// TIA Portal project "ISA_P6" (V16)

(* hardware
DEVICE "SINAMICS G_1"  Sinamics.Device
   slot 0: "Accionamiento_1"  G120 CU250S-2 PN Vector  6SL3246-0BA22-1FA0  4.7.10
      slot 1: "Interfaz PROFINET"  MDD-SinamicsG120-P
   slot 0: "	_0"  Rail  SinamicsG120SVecto
   slot 3: "PM240 IP20"  PM240 IP20  6SL3224-0BE13-7UA0  -
DEVICE "S7-1200 station_1"  S7-1200 Station
   slot 0: "Rack_0"  S7-1200 Rack  Rack  V1.0
   slot 1: "PLC_1"  CPU 1215C DC/DC/DC  6ES7 215-1AG40-0XB0  V4.4
DEVICE "PC-System_1"  SIMATIC PC station
   slot 0: "Estación PC SIMATIC"  Rail  SIMATIC PC-Station  V1.0
      slot 125: "Stationmanager"  Station_Manager  V6.0.4
   slot 1: "HMI_RT_1"  WinCC RT Advanced  6AV2 104-0xxxx-xxxx  16.0.0.0
      slot 33792: "Interfaz del equipo"  Host interface
   slot 2: "IE general_1"  IE General  IE_CP  V8.2.0
*)

// ===== PLC "PLC_1"  CPU 1215C DC/DC/DC =====

VAR_GLOBAL   // PLC tag table "Tabla de variables estándar"
   "ConexiónMotor" AT %Q0.0 : Bool;
   "InversionSentido" AT %Q0.1 : Bool;
   "ConsignaVelocidad" AT %QW64 : Int;
   "ConsignaVelocidadAlcanzada" AT %I0.0 : Bool;
   "ActivarJog1" AT %Q0.2 : Bool;
   "VelocidadActual" AT %IW64 : Word;
END_VAR

DATA_BLOCK "Variables"   // DB1
{ S7_Optimized_Access := 'TRUE' }
VERSION : 0.1
   VAR
      ConexionMotorScada : Bool;
      VelocidadConsignaAlcanzadaScada : Bool;
      InversionMotorScada : Bool;
      VelocidadActualScada : Bool;
      ActivarJog1Scada : Bool;
      VelocidadMotorScada : Int;
      VelocidadNormalizada : Real;
      VelocidadEscalada : Int;
      VelocidadReal : Real;
   END_VAR
BEGIN
END_DATA_BLOCK

DATA_BLOCK "VelocidadReal"   // DB2
{ S7_Optimized_Access := 'TRUE' }
VERSION : 0.1
// stored: InstanceOfName Analog_IN
"Analog_IN"
BEGIN
END_DATA_BLOCK

DATA_BLOCK "Telerruptor_DB"   // DB3
{ S7_Optimized_Access := 'TRUE' }
VERSION : 0.1
// stored: InstanceOfName Telerruptor
"Telerruptor"
BEGIN
END_DATA_BLOCK

DATA_BLOCK "Analog_IN_1_DB"   // DB4
{ S7_Optimized_Access := 'TRUE' }
VERSION : 0.1
// stored: InstanceOfName Analog_IN_1
"Analog_IN_1"
BEGIN
END_DATA_BLOCK

DATA_BLOCK "Analog_OUT_DB"   // DB5
{ S7_Optimized_Access := 'TRUE' }
VERSION : 0.1
// stored: InstanceOfName Analog_OUT
"Analog_OUT"
BEGIN
END_DATA_BLOCK

FUNCTION_BLOCK "Telerruptor"   // FB2, LAD
{ S7_Optimized_Access := 'TRUE' }
VERSION : 0.1
   VAR_INPUT
      Pulsador : Bool;
   END_VAR
   VAR_OUTPUT
      Salida : Bool;
   END_VAR
   VAR
      Flanco : Bool;
      "on/off" : Bool;
      state : Bool;
   END_VAR
   VAR_TEMP   // added for the SCL form of the ladder/FBD networks
      _w1 : Bool;
   END_VAR
BEGIN

REGION Network 1
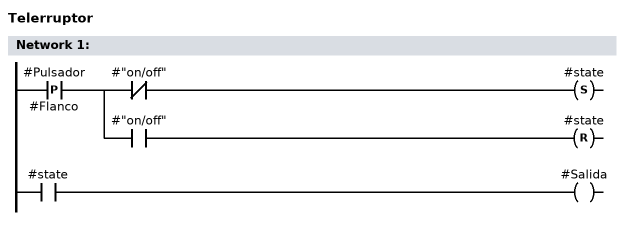
   RUNG wire#powerrail
      P_Contact(operand := #Pulsador, bit := #Flanco)
      wire#w1
      I_Contact( #"on/off" )
      S_Coil( #state )
   END_RUNG
   RUNG wire#w1
      Contact( #"on/off" )
      R_Coil( #state )
   END_RUNG
   RUNG wire#powerrail
      Contact( #state )
      Coil( #Salida )
   END_RUNG
   // the same network as SCL:
   #_w1 := #Pulsador AND NOT #Flanco;   // rising edge of #Pulsador
   #Flanco := #Pulsador;
   IF #_w1 AND NOT #"on/off" THEN #state := TRUE; END_IF;
   IF #_w1 AND #"on/off" THEN #state := FALSE; END_IF;
   #Salida := #state;
END_REGION
END_FUNCTION_BLOCK

FUNCTION_BLOCK "Analog_IN"   // FB4, LAD
{ S7_Optimized_Access := 'TRUE' }
VERSION : 0.1
   VAR_INPUT
      Input : Int;
      X_min : Real;
      X_max : Real;
      Y_min : Real;
      Y_max : Real;
      IsTension : Bool;
   END_VAR
   VAR_OUTPUT
      Output : Real;
   END_VAR
   VAR
      X_min_bits : Int;
      X_max_bits : Int;
      norm : Real;
   END_VAR
   VAR CONSTANT
      tension_pendent : Real := 2764.8;
      intensity_pendent : Real := 1382.4;
   END_VAR
BEGIN

REGION Network 1 (SCL)

   IF #IsTension THEN
       #X_min_bits := REAL_TO_INT(#X_min * #tension_pendent);
       #X_max_bits := REAL_TO_INT(#X_max * #tension_pendent);
   ELSE
       #X_min_bits := REAL_TO_INT(#X_min * #intensity_pendent);
       #X_max_bits := REAL_TO_INT(#X_max * #intensity_pendent);
   END_IF;
END_REGION

REGION Network 2
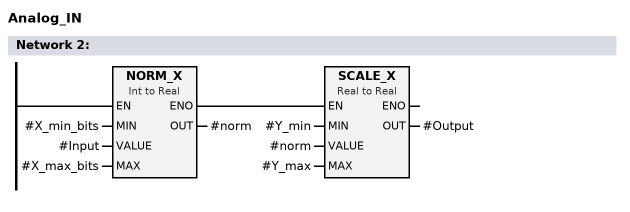
   RUNG wire#powerrail
      { S7_Templates := "[SrcType := Int, DestType := Real]" } Normalize(min := #X_min_bits, value := #Input, max := #X_max_bits, out => #norm)
      { S7_Templates := "[SrcType := Real, DestType := Real]" } Scale(min := #Y_min, value := #norm, max := #Y_max, out => #Output)
   END_RUNG
   // the same network as SCL:
   #norm := NORM_X(MIN := #X_min_bits, VALUE := #Input, MAX := #X_max_bits);
   #Output := SCALE_X(MIN := #Y_min, VALUE := #norm, MAX := #Y_max);
END_REGION
END_FUNCTION_BLOCK

FUNCTION_BLOCK "Analog_IN_1"   // FB4, LAD
{ S7_Optimized_Access := 'TRUE' }
VERSION : 0.1
   VAR_INPUT
      Input : Int;
      X_min : Real;
      X_max : Real;
      Y_min : Real;
      Y_max : Real;
      IsTension : Bool;
   END_VAR
   VAR_OUTPUT
      Output : Real;
   END_VAR
   VAR
      X_min_bits : Int;
      X_max_bits : Int;
      norm : Real;
   END_VAR
   VAR CONSTANT
      tension_pendent : Real := 2764.8;
      intensity_pendent : Real := 1382.4;
   END_VAR
BEGIN

REGION Network 1 (SCL)

   IF #IsTension THEN
       #X_min_bits := REAL_TO_INT(#X_min * #tension_pendent);
       #X_max_bits := REAL_TO_INT(#X_max * #tension_pendent);
   ELSE
       #X_min_bits := REAL_TO_INT(#X_min * #intensity_pendent);
       #X_max_bits := REAL_TO_INT(#X_max * #intensity_pendent);
   END_IF;
END_REGION

REGION Network 2
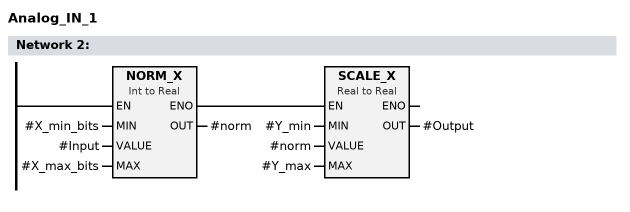
   RUNG wire#powerrail
      { S7_Templates := "[SrcType := Int, DestType := Real]" } Normalize(min := #X_min_bits, value := #Input, max := #X_max_bits, out => #norm)
      { S7_Templates := "[SrcType := Real, DestType := Real]" } Scale(min := #Y_min, value := #norm, max := #Y_max, out => #Output)
   END_RUNG
   // the same network as SCL:
   #norm := NORM_X(MIN := #X_min_bits, VALUE := #Input, MAX := #X_max_bits);
   #Output := SCALE_X(MIN := #Y_min, VALUE := #norm, MAX := #Y_max);
END_REGION
END_FUNCTION_BLOCK

FUNCTION_BLOCK "Analog_OUT"   // FB5, LAD
{ S7_Optimized_Access := 'TRUE' }
VERSION : 0.1
   VAR_INPUT
      Input : Real;
      X_min : Real;
      X_max : Real;
      Y_min : Real;
      Y_max : Real;
      IsTension : Bool;
   END_VAR
   VAR_OUTPUT
      Output : Int;
   END_VAR
   VAR
      Y_min_bits : Int;
      Y_max_bits : Int;
      norm : Real;
   END_VAR
   VAR CONSTANT
      tension_pendent : Real := 2764.8;
      intensity_pendent : Real := 1382.4;
   END_VAR
BEGIN

REGION Network 1 (SCL)

   IF #IsTension THEN
       #Y_min_bits := REAL_TO_INT(#Y_min * #tension_pendent);
       #Y_max_bits := REAL_TO_INT(#Y_max * #tension_pendent);
   ELSE
       #Y_min_bits := REAL_TO_INT(#Y_min * #intensity_pendent);
       #Y_max_bits := REAL_TO_INT(#Y_max * #intensity_pendent);
   END_IF;
END_REGION

REGION Network 2
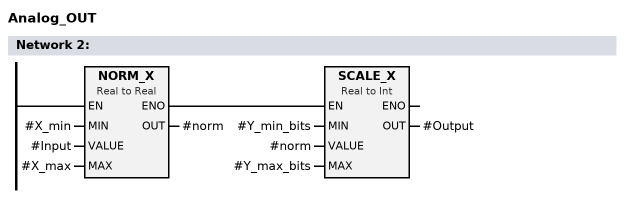
   RUNG wire#powerrail
      { S7_Templates := "[SrcType := Real, DestType := Real]" } Normalize(min := #X_min, value := #Input, max := #X_max, out => #norm)
      { S7_Templates := "[SrcType := Real, DestType := Int]" } Scale(min := #Y_min_bits, value := #norm, max := #Y_max_bits, out => #Output)
   END_RUNG
   // the same network as SCL:
   #norm := NORM_X(MIN := #X_min, VALUE := #Input, MAX := #X_max);
   #Output := SCALE_X(MIN := #Y_min_bits, VALUE := #norm, MAX := #Y_max_bits);
END_REGION
END_FUNCTION_BLOCK

ORGANIZATION_BLOCK "Variador"   // OB1, LAD, ProgramCycle
TITLE = "Main Program Sweep (Cycle)"
{ S7_Optimized_Access := 'TRUE' }
VERSION : 0.1
   VAR_INPUT
      Initial_Call : Bool;   // Initial call of this OB
      Remanence : Bool;   // =True, if remanent data are available
   END_VAR
BEGIN

REGION Network 1
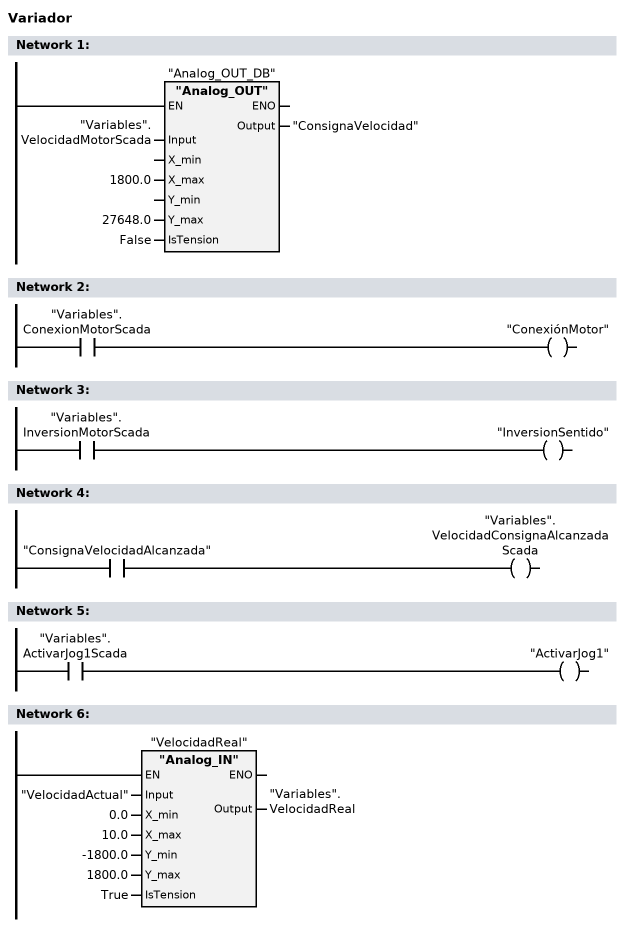
   RUNG wire#powerrail
      "Analog_OUT_DB"(Input := "Variables".VelocidadMotorScada, X_min :=, X_max := 1800.0, Y_min :=, Y_max := 27648.0, IsTension := False, Output => "ConsignaVelocidad")
   END_RUNG
   // the same network as SCL:
   "Analog_OUT_DB"(Input := "Variables".VelocidadMotorScada,   // "Analog_OUT"
                   X_max := 1800.0,
                   Y_max := 27648.0,
                   IsTension := False,
                   Output => "ConsignaVelocidad");
END_REGION

REGION Network 2
   RUNG wire#powerrail
      Contact( "Variables".ConexionMotorScada )
      Coil( "ConexiónMotor" )
   END_RUNG
   // the same network as SCL:
   "ConexiónMotor" := "Variables".ConexionMotorScada;
END_REGION

REGION Network 3
   RUNG wire#powerrail
      Contact( "Variables".InversionMotorScada )
      Coil( "InversionSentido" )
   END_RUNG
   // the same network as SCL:
   "InversionSentido" := "Variables".InversionMotorScada;
END_REGION

REGION Network 4
   RUNG wire#powerrail
      Contact( "ConsignaVelocidadAlcanzada" )
      Coil( "Variables".VelocidadConsignaAlcanzadaScada )
   END_RUNG
   // the same network as SCL:
   "Variables".VelocidadConsignaAlcanzadaScada := "ConsignaVelocidadAlcanzada";
END_REGION

REGION Network 5
   RUNG wire#powerrail
      Contact( "Variables".ActivarJog1Scada )
      Coil( "ActivarJog1" )
   END_RUNG
   // the same network as SCL:
   "ActivarJog1" := "Variables".ActivarJog1Scada;
END_REGION

REGION Network 6
   RUNG wire#powerrail
      "VelocidadReal"(Input := "VelocidadActual", X_min := 0.0, X_max := 10.0, Y_min := -1800.0, Y_max := 1800.0, IsTension := True, Output => "Variables".VelocidadReal)
   END_RUNG
   // the same network as SCL:
   "VelocidadReal"(Input := "VelocidadActual",   // "Analog_IN"
                   X_min := 0.0,
                   X_max := 10.0,
                   Y_min := -1800.0,
                   Y_max := 1800.0,
                   IsTension := True,
                   Output => "Variables".VelocidadReal);
END_REGION
END_ORGANIZATION_BLOCK

(* ===== HMI "HMI_RT_1" =====
system functions are stored by id; their names below are inferred from use
connection "HMI_Conexión_1": ETHERNET, S7_1200_OMS

HMI tags "Tabla de variables estándar"
   "Variables_AvanceMotorScada" : Bool = PLC Variables.ConexionMotorScada, 1 s
   "Variables_RetrocesoMotorScada" : Bool = PLC Variables.InversionMotorScada, 1 s
   "Variables_VelocidadMotorScada" : Int = PLC Variables.VelocidadMotorScada, 1 s
   "Variables_VelocidadConsignaAlcanzada" : Bool = PLC Variables.VelocidadConsignaAlcanzadaScada, 1 s
   "Variables_ActivarJog1Scada" : Bool = PLC Variables.ActivarJog1Scada, 1 s
   "Variables_VelocidadReal" : Real = PLC Variables.VelocidadReal, 1 s

screen "Imagen_1" 800x600
   Button "Botón_1" at 89,271 size 96x32; TextOff 'Conexión'
      on Click: InvertBit("Variables_AvanceMotorScada")
   TextField "Campo de texto_1" at 263,109 size 135x22; Text 'Velocidad'
   Slider "Deslizador_1" at 263,149 size 80x339; Caption 'SIMATIC'
      ProcessValue <- "Variables_VelocidadMotorScada"
   Circle "Círculo_1" at 443,239 size 48x48
      Appearance <- "Variables_VelocidadConsignaAlcanzada"
   TextField "Campo de texto_2" at 356,181 size 214x55; Text 'Velocidad Consigna Alcanzada'
   TextField "Campo de texto_3" at 48,236 size 198x22; Text 'Movimiento Motor'
   Button "Botón_3" at 606,250 size 74x32; TextOff 'JOG1'
      on Press: SetBit("Variables_ActivarJog1Scada")
      on Release: ResetBit("Variables_ActivarJog1Scada")
   TextField "Campo de texto_4" at 537,179 size 201x57; Text 'Activar JOG1 v = 400rpm'
   IOField "Campo ES_1" at 482,415 size 131x32; FormatPattern s9999.99; Unit rpm
      ProcessValue <- "Variables_VelocidadReal"
   TextField "Campo de texto_5" at 483,378 size 263x22; Text 'Velocidad Actual'
   Switch "Interruptor_1" at 82,323 size 120x88; CaptionText 'Inversión'; TextOff 'OFF'; TextOn 'ON'
      ProcessValue <- "Variables_RetrocesoMotorScada"
*)